Fanuc KAREL source: kt00992.KL

-- PROVISIONAL review KL for V940-1; original PC SHA256 6249210a5d349d14708617a5f9f9bd8e9267a397f1439ee7020c8646c209fc26
-- Incomplete behavior may be omitted. Consult companion uncertainty JSON. Do not deploy.
PROGRAM KT00992
%NOLOCKGROUP
VAR
  X : REAL
  Y : REAL
  Z : REAL
  W : REAL
  P : REAL
  R : REAL
-- UNRESOLVED_DECL P1 type=000102
-- UNRESOLVED_DECL P2 type=000102
-- UNRESOLVED_DECL CFG type=00001c
BEGIN
  -- V9_ZERO_TABLE_METADATA_HINT layout=0001; no indexed target words; source/name/runtime held
  -- UNRESOLVED_PC offsets 5-20; opcodes 2E,22,32,35
  -- UNRESOLVED_PC offsets 25-40; opcodes 2E,22,32,35
  -- UNRESOLVED_PC offsets 45-60; opcodes 2E,22,32,35
  -- UNRESOLVED_PC offsets 65-80; opcodes 2E,22,32,35
  -- UNRESOLVED_PC offsets 85-142; opcodes 27,22,1C,22,22,22,22,22,22,22,76
  -- UNRESOLVED_PC offsets 147-151; opcodes 7F
END KT00992
